# EPICS autosave request: xx_auto_saveData_settings.req
$(P)saveData_fileSystem
$(P)saveData_subDir
$(P)saveData_scanNumber
$(P)saveData_realTime1D
